ABB RobotStudio station: robot3gyak.rspag

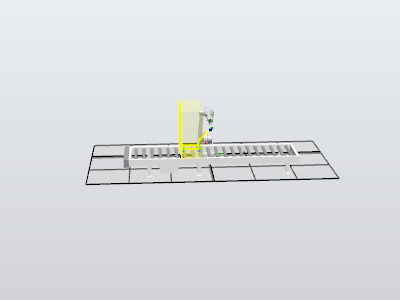
--- station ---
Station robot3gyak (saved by RobotStudio 25.3.11371.0)
Controller IRB1600_10_145, task T_ROB1: task frame (RAPID world) sits at (1500, -740, 435) mm, rotated rx 0 ry 0 rz 90 deg in the station
Controller IRB1600_10_145
  mechanical unit ROB_1: IRB1600_10_145__02, 6 joints, base frame (740, 1500, -435) mm, rotated rx 0 ry 0 rz -90 deg
  mechanical unit CNV1: ?, 1 joints, base frame (0, 0, 0) mm
Layout (positions relative to the parent item):
  - IRB1600_10_145__02 [mechanism, from %ABB.RobotStudio.Models.IRB1600%\IRB1600_10_145_G_02.rslib] at (0, 0, 0) mm; joint values [0, 0, 0, 0, 0.5236, 0] (rad or m)
  - MyTool [mechanism, from Training Objects\myTool.rslib] at (806.29, 0, 1154) mm, rotated rx 180 ry 60 rz 180 deg
  - Conveyor [conveyor]
    - 950_4000_h2 [part] at (1500, -2000, 0) mm, rotated rx 0 ry 0 rz 90 deg, size 4244 x 1170 x 435 mm
    - Curve_thing [part, from Training Objects\Curve_Thing.rslib] at (944.38, 149.94, 667.04) mm, rotated rx 0 ry -5.23 rz 7.04 deg
  - SmartComponent_1 [smart component]
      connections:
        LineSensor.SensorOut -> ConveyorControl.Stop
    - ConveyorControl [smart component, from Components\ConveyorControl.rslib]
        properties: Conveyor=Conveyor
    - LineSensor [smart component, from Components\LineSensor.rslib]
        properties: Start=[0 0 0]; End=[0 0 0.1]; Length=0.1; Radius=0; Tag=(none); SenseMultiple=false; SensedPart=(none); SensedPoint=[0 0 0]
      - _sensorPart_ [part, from Components\LineSensor.rslib]
Attachment: MyTool is attached to IRB1600_10_145__02 / Link6
Conveyor tracking Connection: unit CNV1, TravelOffset=1.2, QueueTrackDistance=0, StartWindowWidth=0.5, SyncSeparation=0, CountsPerMeter=10000
Targets, tools, work objects and paths stored in the station and not in the controller backup, written as RAPID:
! task T_ROB1
MODULE Module1
  CONST robtarget Target_60:=[[449.998977661,699.995788574,90],[0,0.707106781,0.707106781,0],[0,0,0,0],[9E+09,9E+09,9E+09,9E+09,9E+09,0]];
  CONST robtarget Target_70:=[[449.998977661,699.995788574,190],[0,0.707106781,0.707106781,0],[0,0,0,0],[9E+09,9E+09,9E+09,9E+09,9E+09,0]];
ENDMODULE


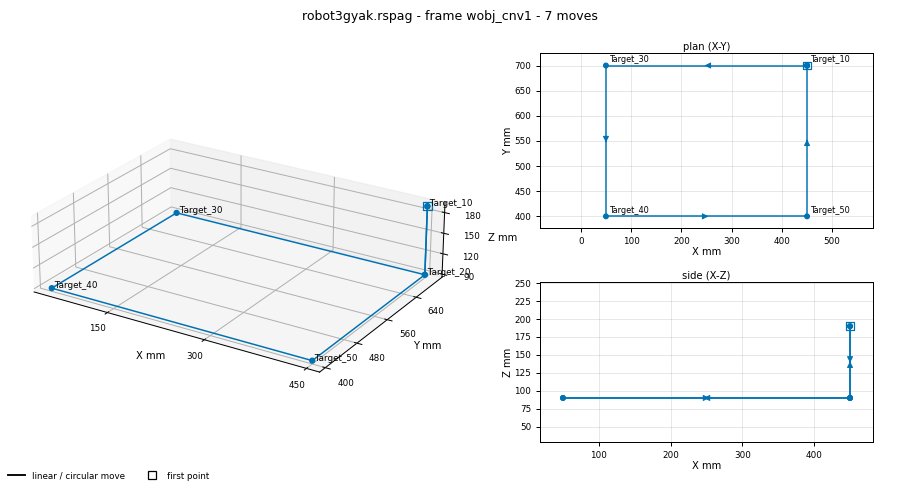
[picture p0: tool path of robot3gyak.rspag in frame wobj_cnv1, 7 of 9 moves have a stored position in this frame; points joined in program order, loops and branches not executed]
--- Controller Data/IRB1600_10_145/RAPID/TASK1/PROGMOD/CalibData.mod ---
MODULE CalibData
    PERS tooldata MyTool:=[TRUE,[[31.792631019,0,229.638935148],[0.945518576,0,0.325568154,0]],[1,[0,0,1],[1,0,0,0],0,0,0]];
    TASK PERS wobjdata wobj_cnv1:=[FALSE,FALSE,"CNV1",[[0,0,0],[1,0,0,0]],[[0,0,0],[1,0,0,0]]];
ENDMODULE

--- Controller Data/IRB1600_10_145/RAPID/TASK1/PROGMOD/Module1.mod ---
MODULE Module1
    CONST jointtarget HOME:=[[0,0,0,0,30,0],[9E+09,9E+09,9E+09,9E+09,9E+09,0]];
    CONST robtarget Target_10:=[[449.998977661,699.995788574,190],[0,0.707106781,0.707106781,0],[0,0,0,0],[9E+09,9E+09,9E+09,9E+09,9E+09,0]];
    CONST robtarget Target_20:=[[449.998977661,699.995788574,90],[0,0.707106781,0.707106781,0],[0,0,0,0],[9E+09,9E+09,9E+09,9E+09,9E+09,0]];
    CONST robtarget Target_30:=[[49.998977661,699.995788574,90],[0,0.707106781,0.707106781,0],[0,0,0,0],[9E+09,9E+09,9E+09,9E+09,9E+09,0]];
    CONST robtarget Target_40:=[[49.998977661,399.995788574,90],[0,0.707106781,0.707106781,0],[0,0,0,0],[9E+09,9E+09,9E+09,9E+09,9E+09,0]];
    CONST robtarget Target_50:=[[449.998977661,399.995788574,90],[0,0.707106781,0.707106781,0],[0,0,0,0],[9E+09,9E+09,9E+09,9E+09,9E+09,0]];
    !***********************************************************
    !
    ! Module:  Module1
    !
    ! Description:
    !   <Insert description here>
    !
    ! Author: anlal
    !
    ! Version: 1.0
    !
    !***********************************************************


    !***********************************************************
    !
    ! Procedure main
    !
    !   This is the entry point of your program
    !
    !***********************************************************
    PROC main()
        Path_10;
    ENDPROC
    PROC Path_10()
        ActUnit CNV1;
        ConfL \Off;
        MoveAbsJ HOME,v1000,fine,MyTool;
        WaitWObj wobj_cnv1;
        MoveL Target_10,v1000,z100,MyTool\WObj:=wobj_cnv1;
        MoveL Target_20,v1000,z0,MyTool\WObj:=wobj_cnv1;
        MoveL Target_30,v1000,z0,MyTool\WObj:=wobj_cnv1;
        MoveL Target_40,v1000,z0,MyTool\WObj:=wobj_cnv1;
        MoveL Target_50,v1000,z0,MyTool\WObj:=wobj_cnv1;
        MoveL Target_20,v1000,z0,MyTool\WObj:=wobj_cnv1;
        MoveL Target_10,v1000,z100,MyTool\WObj:=wobj_cnv1;
        MoveAbsJ HOME,v1000,fine,MyTool;
        DropWObj wobj_cnv1;
    ENDPROC
ENDMODULE

--- Controller Data/IRB1600_10_145/SYSPAR/EIO.cfg ---
EIO:CFG_1.0:6:1::
#
INDUSTRIAL_NETWORK:

      -Name "RobICI" -Label "RobICI Network"
#
ROBICI_DEVICE:

      -Name "CTM1" -TrustLevel "InternalDeviceTrustLevel"\
      -VendorName "ABB Robotics" -ProductName "DSQC2000"\
      -Label "Conveyor Tracking Device 1" -Address "0.0.0.0"
#
EIO_SIGNAL:

      -Name "c1Counts" -SignalType "GI" -Device "CTM1"\
      -DeviceMap "Enc1:position"

      -Name "c1CountsPerSec" -SignalType "AI" -Device "CTM1"\
      -DeviceMap "Enc1:velocity"

      -Name "c1TrigVis" -SignalType "DO" -Device "CTM1" -Label "Trig X21 pin 6"\
      -DeviceMap "Digout1:Setpoint"

      -Name "c1TrigAutoMode" -SignalType "DO" -Device "CTM1"\
      -DeviceMap "Cam1:Connect"

      -Name "c1TrigAutoDist" -SignalType "GO" -Device "CTM1"\
      -DeviceMap "Cam1:Interval"

      -Name "c1TrigAutoEncNo" -SignalType "GO" -Device "CTM1"\
      -DeviceMap "Cam1Enc:DeviceNo"

      -Name "c1CntFromEnc" -SignalType "GI" -Device "CTM1"\
      -DeviceMap "Sync1Enc1:Value"

      -Name "c1SoftSync" -SignalType "DO" -Device "CTM1"\
      -DeviceMap "Sync1Enc1:SyncTrig"

      -Name "c1SpeedBandWidth" -SignalType "GI" -Device "CTM1"\
      -DeviceMap "e1_SpeedBandWidth:SetPoint"

      -Name "c1Position" -SignalType "AO" -MaxLog 21474.8 -MaxPhys 1\
      -MaxPhysLimit 1 -MaxBitVal 2147483647 -MinLog -21474.8 -MinPhys -1\
      -MinPhysLimit -1 -MinBitVal -2147483647 -Size 32

      -Name "c1Speed" -SignalType "AO" -MaxLog 21474.8 -MaxPhys 1\
      -MaxPhysLimit 1 -MaxBitVal 2147483647 -MinLog -21474.8 -MinPhys -1\
      -MinPhysLimit -1 -MinBitVal -2147483647 -Size 32

      -Name "c1Connected" -SignalType "DO"

      -Name "c1NullSpeed" -SignalType "DO"

      -Name "c1PassStw" -SignalType "DO"

      -Name "c1NewObjStrobe" -SignalType "DO" -Access "All"

      -Name "c1WaitWObj" -SignalType "DO"

      -Name "c1DropWObj" -SignalType "DO" -Access "All"

      -Name "c1Rem1PObj" -SignalType "DO" -Access "All"

      -Name "c1RemAllPObj" -SignalType "DO" -Access "All"

      -Name "c1CntToEncStr" -SignalType "DO" -Access "All"

      -Name "c1PosInJobQ" -SignalType "DO" -Default 1

      -Name "c1ObjectsInQ" -SignalType "GO" -Size 8

      -Name "c1CntToEnc" -SignalType "GO" -Size 32

--- Controller Data/IRB1600_10_145/SYSPAR/PROC.cfg ---
PROC:CFG_1.0:6:0::
#
CONVEYOR:

      -name "CNV1" -sensor_type "ICI" -use_sensor "ICI1" -adjustment_speed 850\
      -min_dist -600 -max_dist 1200 -correction_vector_ramp_length 5
#
CONVEYOR_ICI_SENSOR:

      -name "ICI1" -connected_signal "c1Connected" -position_signal "c1Position"\
      -velocity_signal "c1Speed" -position_count_signal "c1Counts"\
      -velocity_count_signal "c1CountsPerSec" -null_speed_signal "c1NullSpeed"\
      -wait_wobj_signal "c1WaitWObj" -drop_wobj_signal "c1DropWObj"\
      -rem_all_pobj_signal "c1RemAllPObj" -rem_one_pobj_signal "c1Rem1PObj"\
      -supervise_max_dist_off  -newobj_strobe "c1NewObjStrobe"\
      -count_to_enc_strobe "c1CntToEncStr" -obj_in_queue_signal "c1ObjectsInQ"\
      -count_from_enc "c1CntFromEnc" -count_to_enc "c1CntToEnc"\
      -StartWinWidth 0.5 -speed_filter_bandwidth "c1SpeedBandWidth"
